TYPE ST_ElementInterfaceIn :
(**************************************************************************************
 * 	Application		:	BoxControl Framework
 *	Revision		:	$Revision: 404529 $
 *	Revision date	:	$Date: 2018-04-23 08:21:38 +0200 (Mo., 23 Apr 2018) $
 *	Last changed by	:	$Author: b7bolm $
 *	URL				:	$URL: http://almscdc.swisslog.com/repo/SWPD/Development/BoxControlFramework/20_Release/trunk/01_Software/BCF/BCF/JumpStart/20_Product/10_App/13_Elements/10_Lib/10_Conv/01_DUTs/ST_ElementInterfaceIn.TcDUT $
 *
 *	Purpose			:	Element data
 *
 * ------------------------------------------------------------------------------------
 *	Copyright Swisslog [IP AG], Switzerland. All rights reserved.
 * 
 * ------------------------------------------------------------------------------------
 *	
 * 	Revision History: 
 *
 * 	VERSION			DATE			INITIALS			DESCRIPTION
 *	0.1				01.01.2001		swl					Example
 *
 **************************************************************************************)	
STRUCT
	GroupState			: ST_PositionState;
	FunctionOrders		: ARRAY[1..Conveyor.NUMBER_OF_FUNCTIONS_PER_ELEMENT] OF ST_FunctionOrders;
	ElementStates		: ST_MasterSlaveStates;
	ElementEnable		: BOOL := TRUE; // External function enable 
END_STRUCT
END_TYPE

(* stored: Version 1.1.0.1, ProductVersion 3.1.4022.12
   DUT ST_ElementInterfaceIn: Id {ba286658-fea4-4c34-92da-a9fcc3eadf40} *)
